Fanuc KAREL source: RPOSREG_SEND.kl

PROGRAM T
%NOLOCKGROUP
VAR
 v0 : STRING[40]
 v1 : INTEGER
 v2 : INTEGER
 v3 : INTEGER
 v4 : INTEGER
 v5 : INTEGER
 v6 : INTEGER
BEGIN
 RPOSREG_SEND(v0, v1, v2, v3, v4, v5, v6)
END T
